FUNCTION_BLOCK FB_XPIM_Opal
VAR
	{attribute 'pytmc' := '
		pv: PWR
		ZNAM: OFF
		ONAM: ON
	'}
	bOpalPower AT %Q*: BOOL;
	
	bOpalInit: BOOL := FALSE;
END_VAR

// Turn the Opal on by default
IF NOT bOpalInit THEN
	bOpalPower := TRUE;
	bOpalInit := TRUE;
END_IF

END_FUNCTION_BLOCK

(* stored: Version 1.1.0.1, ProductVersion 3.1.4022.12
   POU FB_XPIM_Opal: Id {b1b890b6-3afe-4a18-b0c8-85c6c6d77f08}, SpecialFunc None *)
